{attribute 'GeneratedUsingTerminal: EL3314-0000-0018'}
{attribute addProperty BoxType "EL3314-0000-0018"}
{attribute addProperty Id "TC_Inputs_Channel_1AT %I*TC_Inputs_Channel_4A3944819TC_Inputs_Channel_2AT %I*TC_Inputs_Channel_4A3944819TC_Inputs_Channel_3AT %I*TC_Inputs_Channel_4A3944819TC_Inputs_Channel_4AT %I*TC_Inputs_Channel_4A3944819WcStateAT %I*WcState_9091E0EB2InfoDataAT %I*InfoData_94A18F5E2"}
{attribute addProperty CRC "2556586545"}
{attribute addProperty Size "40"}
TYPE EL3314_98626A31 EXTENDS EtcSlaveTerminalBase_947E5A46 :
STRUCT
	{attribute addProperty Name "TC_Inputs_Channel_1"}
	TC_Inputs_Channel_1 : TC_Inputs_Channel_4A394481;
	{attribute addProperty Name "TC_Inputs_Channel_2"}
	TC_Inputs_Channel_2 : TC_Inputs_Channel_4A394481;
	{attribute addProperty Name "TC_Inputs_Channel_3"}
	TC_Inputs_Channel_3 : TC_Inputs_Channel_4A394481;
	{attribute addProperty Name "TC_Inputs_Channel_4"}
	TC_Inputs_Channel_4 : TC_Inputs_Channel_4A394481;
	{attribute addProperty Name "WcState"}
	WcState : WcState_9091E0EB;
	{attribute addProperty Name "InfoData"}
	InfoData : InfoData_94A18F5E;
END_STRUCT
END_TYPE

(* stored: Version 1.2.0.0, ProductVersion 3.1.4024.9
   DUT EL3314_98626A31: Id {d790bb9f-fd73-4338-bb53-f59a1a3593ea} *)
